// TIA Portal V20 export
TYPE "typeFDoorSwitchStatus"
// stored: Access Published, IsFailsafeCompliant true, Namespace Safety
   STRUCT
      autoSpliceDoorOpen : Bool;   // F Door Open Status
      unwinderMainDoorOpen : Bool;   // F Door Open Status
      unwinderTopDoorOpen : Bool;   // F Door Open Status
      unwinderBtmDoorOpen : Bool;   // F Door Open Status
      stackTableDoorOpen : Bool;   // F Door Open Status
      jrWinderDoorOpen : Bool;   // F Door Open Status
      anodeWasteDoorOpen : Bool;   // F Door Open Status
      stackTableRearDoorOpen : Bool;   // F Door Open Status
      cathodeWasteDoorOpen : Bool;   // F Door Open Status
      unwinderRearDoorOpen : Bool;   // F Door Open Status
   END_STRUCT;
END_TYPE
